Omron CX-Programmer project NewProject (CX-Programmer 9.66)

# PLC NewPLC1: CP1L-E EM

## Global symbols (name address type ; comment)
0.05 BOOL  ; SQ1-Открытие ворот(ств.ОТКРЫТА)
0.07 BOOL  ; SQ2-Закрытие ворот(ств.ЗАКРЫТА)
0.00 BOOL  ; 0-Ручной/1-Автомат
0.01 BOOL  ; Кнопка открытия (SB10)
0.02 BOOL  ; Кнопка закрытия (SB20)
0.03 BOOL  ; BF1 Радар
0.04 BOOL  ; BQ1 Прострел ворот
0.10 BOOL  ; BQ2 Датчик верхний (с ЦЕХА)
100.02 BOOL  ; Открытие ворот
100.03 BOOL  ; Закрытие ворот
100.04 BOOL  ; $?St$Bk?_#[61] / HA "звуковой сигнал"$?St$Bk?_#[61]
100.05 BOOL  ; $?St$Bk?_#[62] / HL1 ЗЕЛЁНАЯ лампочка "работа"$?St$Bk?_#[62]
100.06 BOOL  ; HL2 ЖЁЛТАЯ лампочка
100.07 BOOL  ; $?St$Bk?_#[63] / КРАСНАЯ лампочка "АВАРИЯ"$?St$Bk?_#[63]
10.02 BOOL  ; Открытие ворот
10.03 BOOL  ; Закрытие ворот
10.04 BOOL  ; $?St$Bk?_#[64] / HA "звуковой сигнал"$?St$Bk?_#[64]
10.05 BOOL  ; $?St$Bk?_#[65] / HL1 ЗЕЛЁНАЯ лампочка "работа"$?St$Bk?_#[65]
10.06 BOOL  ; HL2 ЖЁЛТАЯ лампочка
10.07 BOOL  ; $?St$Bk?_#[66] / КРАСНАЯ лампочка "АВАРИЯ"$?St$Bk?_#[66]
200.00 BOOL  ; Створка ОТКРЫТА
200.01 BOOL  ; Створка ЗАКРЫТА
200.05 BOOL  ; Сигнал на открытие
200.06 BOOL  ; Сигнал на закрытие
200.07 BOOL  ; Если при закрытии сработал датчик BF1/BQ2
200.08 BOOL  ; Цикл закрытия
200.09 BOOL  ; Начало таймера на закрытие если не достигла концевика (SB20)
210.00 BOOL  ; Открытие в ручном режиме
210.01 BOOL  ; Закрытие в ручном режиме
210.04 BOOL  ; Звонок при открытии
210.10 BOOL  ; АВАРИЯ
211.00 BOOL  ; открытие при пересечении BQ1 когда ворота закрывались
212.00 BOOL  ; если пересекут во время закрытия ворот датчик BQ1
213.00 BOOL  ; Открытие ворот если пересекли датчик BQ1 о время закрытия ворот
T0000 BOOL  ; Таймер перед закрытием
T0001 BOOL  ; Таймер по истечению которого подается сигнал на аварию
T0003 BOOL  ; Задержка перед открытием
T0004 BOOL  ; Начало таймера на закрытие если не достигла концевика (SB20)
T0005 BOOL  ; Таймер перед открытием ворот если кто-то пересек BQ1 когда ворота закрывались

## Program NewProgram1 (cyclic task 0)

### Section Section1

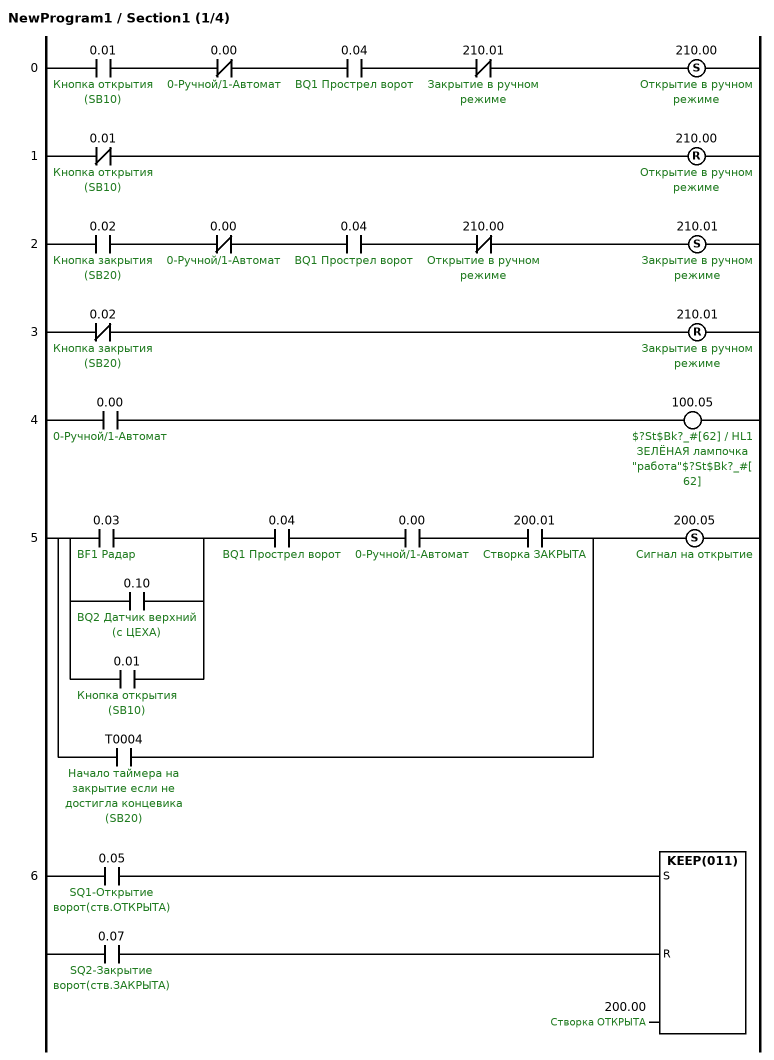
; rung 0
LD 0.01  ; Кнопка открытия (SB10)
ANDNOT 0.00  ; 0-Ручной/1-Автомат
AND 0.04  ; BQ1 Прострел ворот
ANDNOT 210.01  ; Закрытие в ручном режиме
SET 210.00  ; Открытие в ручном режиме
; rung 1
LDNOT 0.01  ; Кнопка открытия (SB10)
RSET 210.00  ; Открытие в ручном режиме
; rung 2
LD 0.02  ; Кнопка закрытия (SB20)
ANDNOT 0.00  ; 0-Ручной/1-Автомат
AND 0.04  ; BQ1 Прострел ворот
ANDNOT 210.00  ; Открытие в ручном режиме
SET 210.01  ; Закрытие в ручном режиме
; rung 3
LDNOT 0.02  ; Кнопка закрытия (SB20)
RSET 210.01  ; Закрытие в ручном режиме
; rung 4
LD 0.00  ; 0-Ручной/1-Автомат
OUT 100.05  ; $?St$Bk?_#[62] / HL1 ЗЕЛЁНАЯ лампочка "работа"$?St$Bk?_#[62]
; rung 5
LD 0.03  ; BF1 Радар
OR 0.10  ; BQ2 Датчик верхний (с ЦЕХА)
OR 0.01  ; Кнопка открытия (SB10)
AND 0.04  ; BQ1 Прострел ворот
AND 0.00  ; 0-Ручной/1-Автомат
AND 200.01  ; Створка ЗАКРЫТА
OR T0004  ; Начало таймера на закрытие если не достигла концевика (SB20)
SET 200.05  ; Сигнал на открытие
; rung 6
LD 0.05  ; SQ1-Открытие ворот(ств.ОТКРЫТА)
LD 0.07  ; SQ2-Закрытие ворот(ств.ЗАКРЫТА)
KEEP(011) 200.00  ; Створка ОТКРЫТА

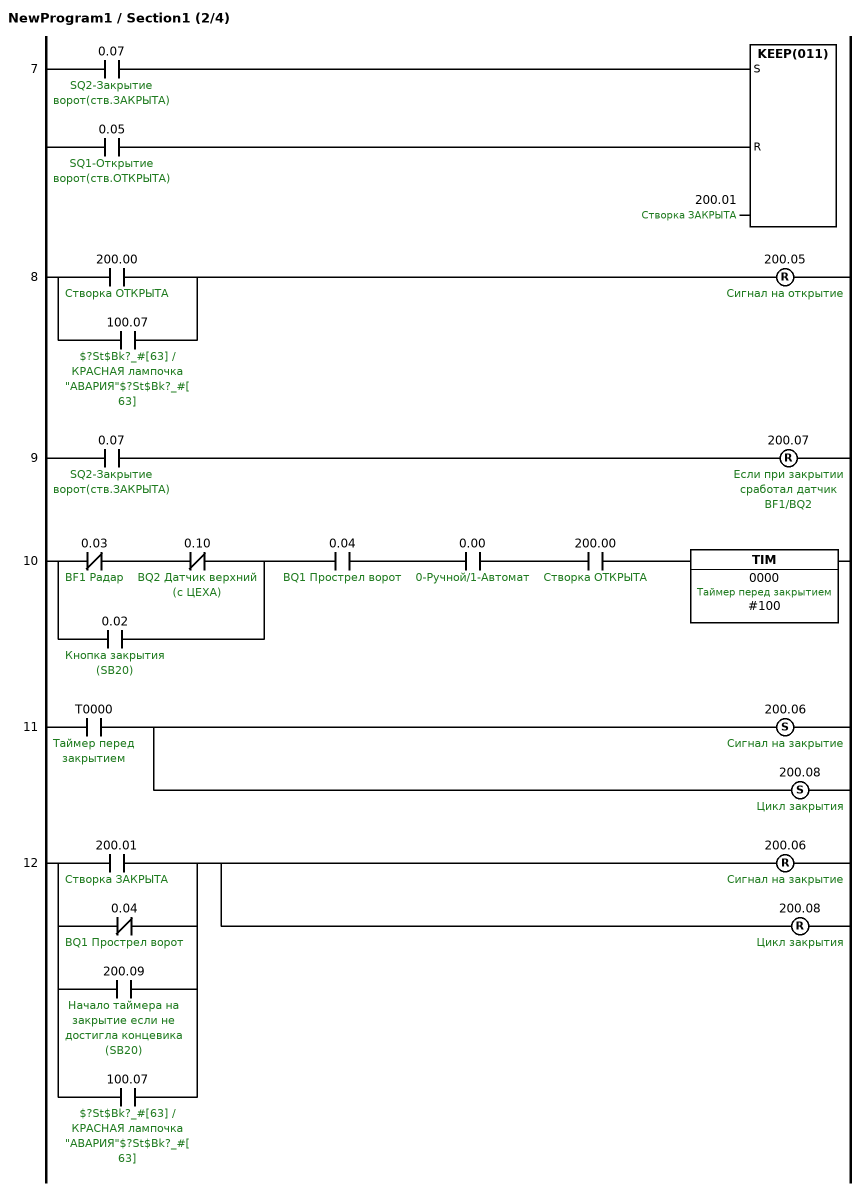
; rung 7
LD 0.07  ; SQ2-Закрытие ворот(ств.ЗАКРЫТА)
LD 0.05  ; SQ1-Открытие ворот(ств.ОТКРЫТА)
KEEP(011) 200.01  ; Створка ЗАКРЫТА
; rung 8
LD 200.00  ; Створка ОТКРЫТА
OR 100.07  ; $?St$Bk?_#[63] / КРАСНАЯ лампочка "АВАРИЯ"$?St$Bk?_#[63]
RSET 200.05  ; Сигнал на открытие
; rung 9
LD 0.07  ; SQ2-Закрытие ворот(ств.ЗАКРЫТА)
RSET 200.07  ; Если при закрытии сработал датчик BF1/BQ2
; rung 10
LDNOT 0.03  ; BF1 Радар
ANDNOT 0.10  ; BQ2 Датчик верхний (с ЦЕХА)
OR 0.02  ; Кнопка закрытия (SB20)
AND 0.04  ; BQ1 Прострел ворот
AND 0.00  ; 0-Ручной/1-Автомат
AND 200.00  ; Створка ОТКРЫТА
TIM 0000 #100  ; Таймер перед закрытием
; rung 11
LD T0000  ; Таймер перед закрытием
SET 200.06  ; Сигнал на закрытие
SET 200.08  ; Цикл закрытия
; rung 12
LD 200.01  ; Створка ЗАКРЫТА
ORNOT 0.04  ; BQ1 Прострел ворот
OR 200.09  ; Начало таймера на закрытие если не достигла концевика (SB20)
OR 100.07  ; $?St$Bk?_#[63] / КРАСНАЯ лампочка "АВАРИЯ"$?St$Bk?_#[63]
RSET 200.06  ; Сигнал на закрытие
RSET 200.08  ; Цикл закрытия

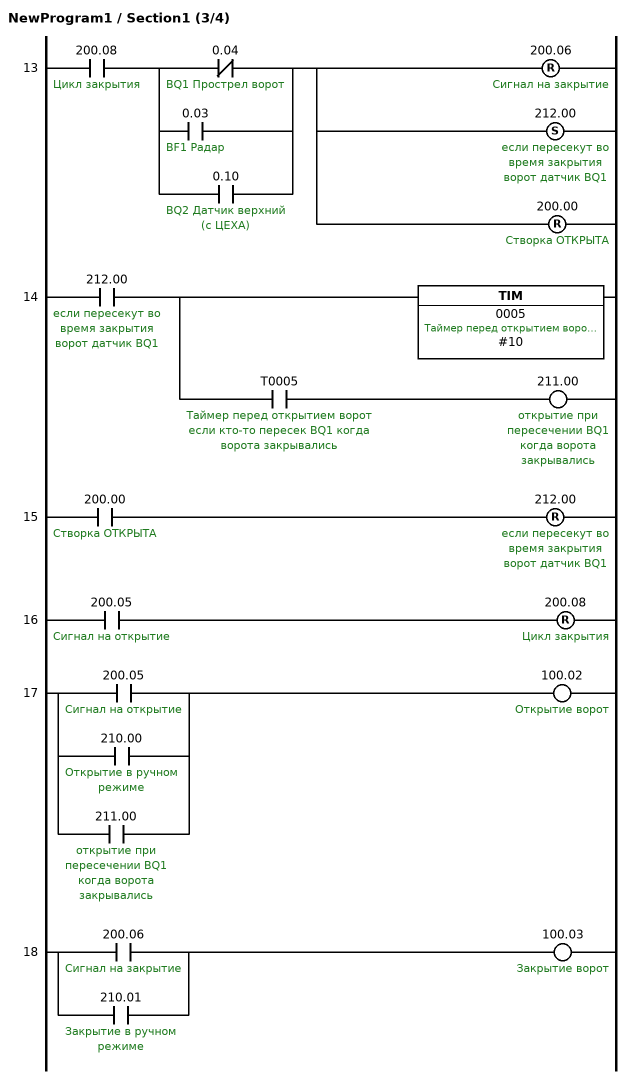
; rung 13
LD 200.08  ; Цикл закрытия
LDNOT 0.04  ; BQ1 Прострел ворот
OR 0.03  ; BF1 Радар
OR 0.10  ; BQ2 Датчик верхний (с ЦЕХА)
ANDLD
RSET 200.06  ; Сигнал на закрытие
SET 212.00  ; если пересекут во время закрытия ворот датчик BQ1
RSET 200.00  ; Створка ОТКРЫТА
; rung 14
LD 212.00  ; если пересекут во время закрытия ворот датчик BQ1
TIM 0005 #10  ; Таймер перед открытием ворот если кто-то пересек BQ1 когда ворота закрывались
AND T0005  ; Таймер перед открытием ворот если кто-то пересек BQ1 когда ворота закрывались
OUT 211.00  ; открытие при пересечении BQ1 когда ворота закрывались
; rung 15
LD 200.00  ; Створка ОТКРЫТА
RSET 212.00  ; если пересекут во время закрытия ворот датчик BQ1
; rung 16
LD 200.05  ; Сигнал на открытие
RSET 200.08  ; Цикл закрытия
; rung 17
LD 200.05  ; Сигнал на открытие
OR 210.00  ; Открытие в ручном режиме
OR 211.00  ; открытие при пересечении BQ1 когда ворота закрывались
OUT 100.02  ; Открытие ворот
; rung 18
LD 200.06  ; Сигнал на закрытие
OR 210.01  ; Закрытие в ручном режиме
OUT 100.03  ; Закрытие ворот

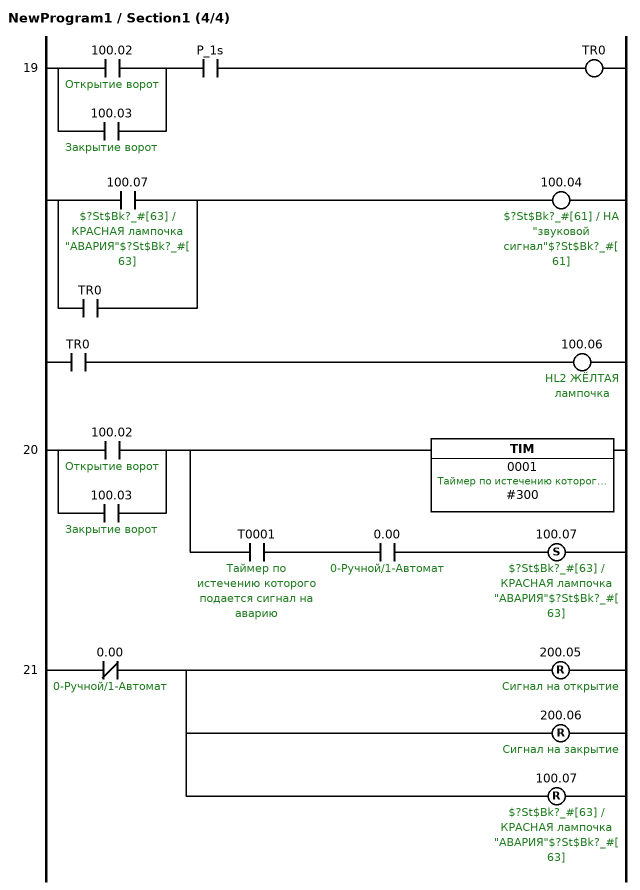
; rung 19
LD 100.07  ; $?St$Bk?_#[63] / КРАСНАЯ лампочка "АВАРИЯ"$?St$Bk?_#[63]
LD 100.02  ; Открытие ворот
OR 100.03  ; Закрытие ворот
AND P_1s
OUT TR0
ORLD
OUT 100.04  ; $?St$Bk?_#[61] / HA "звуковой сигнал"$?St$Bk?_#[61]
LD TR0
OUT 100.06  ; HL2 ЖЁЛТАЯ лампочка
; rung 20
LD 100.02  ; Открытие ворот
OR 100.03  ; Закрытие ворот
TIM 0001 #300  ; Таймер по истечению которого подается сигнал на аварию
AND T0001  ; Таймер по истечению которого подается сигнал на аварию
AND 0.00  ; 0-Ручной/1-Автомат
SET 100.07  ; $?St$Bk?_#[63] / КРАСНАЯ лампочка "АВАРИЯ"$?St$Bk?_#[63]
; rung 21
LDNOT 0.00  ; 0-Ручной/1-Автомат
RSET 200.05  ; Сигнал на открытие
RSET 200.06  ; Сигнал на закрытие
RSET 100.07  ; $?St$Bk?_#[63] / КРАСНАЯ лампочка "АВАРИЯ"$?St$Bk?_#[63]

### Section END
; rung 0
END(001)